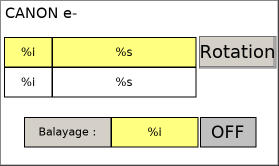
VISUALIZATION SA_EVAP  // 279x166
VAR_IN_OUT
	m_Input_Crucible:   BLOCK_IND_CR_396_TELEMARK;
	m_Input_Sweep:		BLOCK_TELEMARK_CHEETAH_SWEEP;	
END_VAR
    RoundedRectangle (0,0 279x166), text variable: m_Input_Crucible.MNEMO
    Rectangle (2,1 104x24), "CANON e-"
    Rectangle (111,117 87x30), "%i", text variable: m_Input_Sweep.PRM_NbBal, input disabled if: NOT (Global_Variables.PRG_USER.ACTU_USER.FONCTION_SA AND NOT MACHINE.STATE_PROD)
        OnMouseClick: write the text variable via InputWithLimits, min 1, max 8
    Rectangle (24,117 87x30), "Balayage :"
    Rectangle (4,37 48x30), "%i", text variable: m_Input_Crucible.PRM_NCR, input disabled if: NOT (Global_Variables.PRG_USER.ACTU_USER.FONCTION_SA AND NOT MACHINE.STATE_PROD)
        OnMouseClick: write the text variable via InputWithLimits, min 1, max m_Input_Crucible.CONF_NCR
    Rectangle (52,37 144x30), "%s", text variable: m_Input_Crucible.PRM_MAT[m_Input_Crucible.PRM_NCR]
    Button (199,36 77x32), "Rotation", input disabled if: NOT (PRG_USER.ACTU_USER.FONCTION_SA AND NOT MACHINE.STATE_Prod)
        tap PRG_EVAP.PRM_Forcage_Crucible
    RoundedRectangle (200,117 56x30), "ON", invisible if: NOT m_Input_Sweep.STATE_ON
    RoundedRectangle (200,117 56x30), "OFF", invisible if: NOT m_Input_Sweep.STATE_OFF
    Rectangle (4,67 48x30), "%i", text variable: m_Input_Crucible.STATE_POS
    Rectangle (52,67 144x30), "%s", text variable: m_Input_Crucible.PRM_MAT[m_Input_Crucible.STATE_POS], invisible if: (m_Input_Crucible.STATE_POS < 1) or (m_Input_Crucible.STATE_POS > m_Input_Crucible.CONF_NCR)
END_VISUALIZATION

(* stored: Version 1.1.0.1, ProductVersion 3.1.4026.18
   Visu SA_EVAP: Id {236221ba-b39d-4741-98a3-94e0837e488b} *)
